# EPICS StreamDevice protocol: protocols/dac_step.proto
Terminator = LF;
ExtraInput = Ignore;

getBQ {
        in "%0d";
}
